FUNCTION Convert_DT_TO_LREAL : Hresult
VAR_INPUT
	in : DT;
	out : REFERENCE TO LREAL;
END_VAR
VAR
	converted : LREAL;
END_VAR

converted := DT_TO_LREAL(in);

IF (LREAL_TO_DT(converted) <> in) THEN
	Convert_DT_TO_LREAL := INCOMPATIBLE;
	RETURN;
END_IF

out := converted;

END_FUNCTION

(* stored: Version 1.1.0.1, ProductVersion 3.1.4024.12
   POU Convert_DT_TO_LREAL: Id {7d1fc577-f57d-4ea6-bd4d-a288d56f66d8}, SpecialFunc None *)
